// TIA Portal project "esteira_rejeito" (V16)
// primeiro projeto para o rejeito

(* hardware
DEVICE "S7-1200 station_1"  S7-1200 Station
   slot 0: "Rack_0"  S7-1200 Rack  Rack  V1.0
   slot 1: "PLC_1"  CPU 1212C DC/DC/DC  6ES7 212-1AE40-0XB0  V4.4
DEVICE "HMI_1"  KTP400 Basic PN
   slot 0: "HMI_1"  KTP400 Basic PN  6AV2 123-2DB03-0AX0  16.0.0.0
   slot 1: "HMI_RT_1"  KTP400 Basic PN  6AV2 123-2DB03-0AX0  16.0.0.0
   slot 5: "HMI_1.IE_CP_1"  PROFINET Interface  16.0.0.0
      slot 1: "PROFINET Interface_1"  PROFINET Interface
         slot 1: "Port_1"  Port
*)

// ===== PLC "PLC_1"  CPU 1212C DC/DC/DC =====

VAR_GLOBAL   // PLC tag table "Default tag table"
   "encoder_bk10_2101" AT %ID1000 : DInt;
   "ativa motor_bk10_2101" AT %M0.1 : Bool;
   "ativa motor_bk10_2101(1)" AT %Q0.0 : Bool;
   "sensor_01" AT %I0.1 : Bool;
   "sensor_02" AT %I0.2 : Bool;
   "set rest" AT %M0.2 : Bool;
   "b1 liga manual" AT %I0.3 : Bool;
   "rej_01" AT %M0.3 : Bool;
   "rej_01(1)" AT %M0.4 : Bool;
   "sensor_04" AT %I0.4 : Bool;
   "sensor_05" AT %I0.5 : Bool;
   "sensor_06" AT %I0.6 : Bool;
   "ativa motor_rej_01" AT %Q0.1 : Bool;
   "ativa motor_rej_02" AT %Q0.2 : Bool;
   "ativa motor_rej_03" AT %Q0.3 : Bool;
   "sinaleiro_L01" AT %Q0.4 : Bool;
   "rej_02" AT %M0.5 : Bool;
   "rej_02(2)" AT %M0.6 : Bool;
   "rej_03" AT %M0.7 : Bool;
   "rej_03(1)" AT %M1.0 : Bool;
END_VAR

// folder: System blocks/Program resources

DATA_BLOCK "db_rej_01"   // DB3
{ S7_Optimized_Access := 'TRUE' }
AUTHOR : Simatic
FAMILY : IEC
NAME : IEC_TMR
VERSION : 1.0
// stored: InstanceOfName IEC_TIMER
"IEC_TIMER"
BEGIN
END_DATA_BLOCK

DATA_BLOCK "db_rej_02"   // DB4
{ S7_Optimized_Access := 'TRUE' }
AUTHOR : Simatic
FAMILY : IEC
NAME : IEC_TMR
VERSION : 1.0
// stored: InstanceOfName IEC_TIMER
"IEC_TIMER"
BEGIN
END_DATA_BLOCK

// folder: (top level)

FUNCTION "fc_bk10_2101" : Void   // FC2, LAD
{ S7_Optimized_Access := 'TRUE' }
VERSION : 0.1
   VAR_INPUT
      Input_1 : DInt;
   END_VAR
BEGIN

REGION Network 1
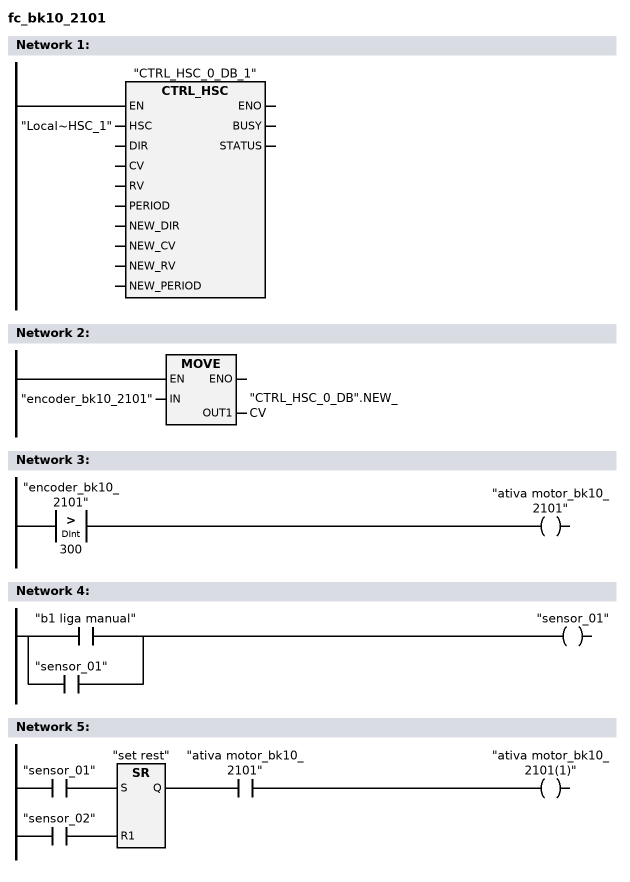
   "CTRL_HSC_0_DB_1"(HSC := "Local~HSC_1");   // CTRL_HSC
END_REGION

REGION Network 2
   RUNG wire#powerrail
      Move(in := "encoder_bk10_2101", out1 => "CTRL_HSC_0_DB".NEW_CV)
   END_RUNG
   // the same network as SCL:
   "CTRL_HSC_0_DB".NEW_CV := "encoder_bk10_2101";
END_REGION

REGION Network 3
   RUNG wire#powerrail
      { S7_Templates := "SrcType := DInt" } GT_Contact(in1 := "encoder_bk10_2101", in2 := 300)
      Coil( "ativa motor_bk10_2101" )
   END_RUNG
   // the same network as SCL:
   "ativa motor_bk10_2101" := "encoder_bk10_2101" > 300;
END_REGION

REGION Network 4
   RUNG wire#powerrail
      Contact( "b1 liga manual" )
      wire#w1
      Coil( "sensor_01" )
   END_RUNG
   RUNG wire#powerrail
      Contact( "sensor_01" )
   END_RUNG wire#w1
   // the same network as SCL:
   "sensor_01" := "b1 liga manual" OR "sensor_01";
END_REGION

REGION Network 5
   RUNG wire#powerrail
      Contact( "sensor_01" )
      S_SR(operand := "set rest", r1 := wire#w1)
      Contact( "ativa motor_bk10_2101" )
      Coil( "ativa motor_bk10_2101(1)" )
   END_RUNG
   RUNG wire#powerrail
      Contact( "sensor_02" )
   END_RUNG wire#w1
   // the same network as SCL:
   IF "sensor_01" THEN
       "set rest" := TRUE;   // SR flip-flop
   END_IF;
   IF "sensor_02" THEN "set rest" := FALSE; END_IF;
   "ativa motor_bk10_2101(1)" := "set rest" AND "ativa motor_bk10_2101";
END_REGION
END_FUNCTION

FUNCTION "fc_rej_01" : Void   // FC3, LAD
{ S7_Optimized_Access := 'TRUE' }
VERSION : 0.1
   VAR_TEMP   // added for the SCL form of the ladder/FBD networks
      _w1 : Bool;
   END_VAR
BEGIN

REGION Network 1
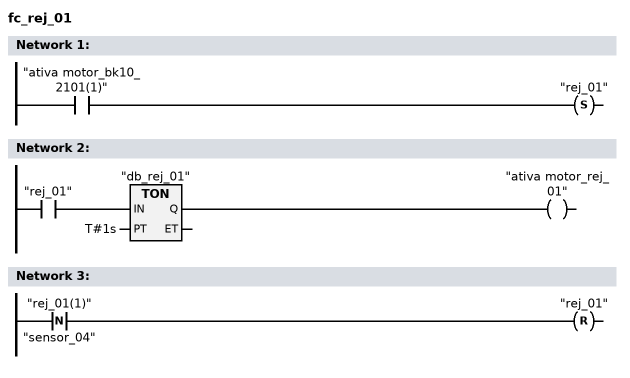
   RUNG wire#powerrail
      Contact( "ativa motor_bk10_2101(1)" )
      S_Coil( "rej_01" )
   END_RUNG
   // the same network as SCL:
   IF "ativa motor_bk10_2101(1)" THEN "rej_01" := TRUE; END_IF;
END_REGION

REGION Network 2
   "db_rej_01".TON(IN := "rej_01", PT := T#1s);
   "ativa motor_rej_01" := "db_rej_01".Q;
END_REGION

REGION Network 3
   RUNG wire#powerrail
      N_Contact(operand := "rej_01(1)", bit := "sensor_04")
      R_Coil( "rej_01" )
   END_RUNG
   // the same network as SCL:
   #_w1 := NOT "rej_01(1)" AND "sensor_04";   // falling edge of "rej_01(1)"
   "sensor_04" := "rej_01(1)";
   IF #_w1 THEN "rej_01" := FALSE; END_IF;
END_REGION
END_FUNCTION

FUNCTION "fc_rej_04" : Void   // FC4, LAD
{ S7_Optimized_Access := 'TRUE' }
VERSION : 0.1
   VAR_TEMP   // added for the SCL form of the ladder/FBD networks
      _w1 : Bool;
   END_VAR
BEGIN

REGION Network 1
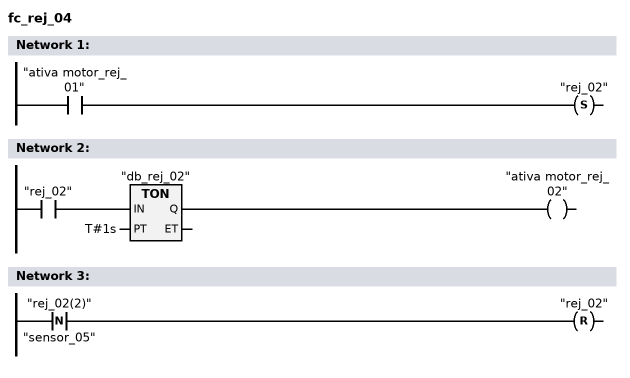
   RUNG wire#powerrail
      Contact( "ativa motor_rej_01" )
      S_Coil( "rej_02" )
   END_RUNG
   // the same network as SCL:
   IF "ativa motor_rej_01" THEN "rej_02" := TRUE; END_IF;
END_REGION

REGION Network 2
   "db_rej_02".TON(IN := "rej_02", PT := T#1s);
   "ativa motor_rej_02" := "db_rej_02".Q;
END_REGION

REGION Network 3
   RUNG wire#powerrail
      N_Contact(operand := "rej_02(2)", bit := "sensor_05")
      R_Coil( "rej_02" )
   END_RUNG
   // the same network as SCL:
   #_w1 := NOT "rej_02(2)" AND "sensor_05";   // falling edge of "rej_02(2)"
   "sensor_05" := "rej_02(2)";
   IF #_w1 THEN "rej_02" := FALSE; END_IF;
END_REGION
END_FUNCTION

ORGANIZATION_BLOCK "Main"   // OB1, LAD, ProgramCycle
TITLE = "Main Program Sweep (Cycle)"
{ S7_Optimized_Access := 'TRUE' }
VERSION : 0.1
   VAR_INPUT
      Initial_Call : Bool;   // Initial call of this OB
      Remanence : Bool;   // =True, if remanent data are available
   END_VAR
BEGIN
END_ORGANIZATION_BLOCK

ORGANIZATION_BLOCK "ob_bk10_2101"   // OB123, LAD, ProgramCycle
TITLE = "Main Program Sweep (Cycle)"
{ S7_Optimized_Access := 'TRUE' }
VERSION : 0.1
   VAR_INPUT
      Initial_Call : Bool;   // Initial call of this OB
      Remanence : Bool;   // =True, if remanent data are available
   END_VAR
BEGIN

REGION Network 1
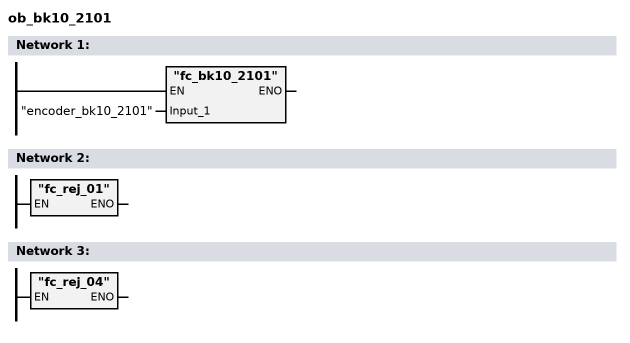
   RUNG wire#powerrail
      "fc_bk10_2101"(Input_1 := "encoder_bk10_2101")
   END_RUNG
   // the same network as SCL:
   "fc_bk10_2101"(Input_1 := "encoder_bk10_2101");
END_REGION

REGION Network 2
   RUNG wire#powerrail
      "fc_rej_01"()
   END_RUNG
   // the same network as SCL:
   "fc_rej_01"();
END_REGION

REGION Network 3
   RUNG wire#powerrail
      "fc_rej_04"()
   END_RUNG
   // the same network as SCL:
   "fc_rej_04"();
END_REGION
END_ORGANIZATION_BLOCK

(* ===== HMI "HMI_RT_1" =====
system functions are stored by id; their names below are inferred from use

HMI tags "Default tag table"
   "Tag_ScreenNumber" : UInt, internal

Template "Template_1" 480x272
   Button "Exit" at 388,227 size 63x44; TextOff 'Exit'; PictureOff "ExitRuntime_KTP400_Basic_PN_TR"; PictureOn "ExitRuntime_KTP400_Basic_PN_TR"
      on Release: StopRuntime(0)
   Button "Template_Button" at 268,227 size 63x44; TextOff 'Text'
   Button "Alarms" at 148,227 size 63x44; TextOff 'Alarms'; PictureOff "AlarmDisplay_KTP400_Basic_PN_TR"; PictureOn "AlarmDisplay_KTP400_Basic_PN_TR"
      on Release: function_ef3f5d25("Alarm window_Unacknowledged", -1)
   Button "Start screen" at 28,227 size 63x44; TextOff 'Start screen'; PictureOff "NavigateHome_KTP400_Basic_PN_TR"; PictureOn "NavigateHome_KTP400_Basic_PN_TR"
      on Release: ActivateScreen("Root screen", 0)
   SymbolicIOField "Symbolic_IO_Field_Screen" at 82,8 size 311x29; TextOff '0'; TextOn '1'; TextList "TextList_ScreenNames"
      ProcessValue <- "Tag_ScreenNumber"
      on Change: ActivateScreenByNumber("Tag_ScreenNumber", 0)
   DateTimeField "HmiScreenItemData" at 395,22 size 85x22
   DateTimeField "HmiScreenItemData_1" at 395,0 size 85x22
   GraphicView "Logo" at 0,0 size 80x45; Picture "Logo of HMI_1"

screen "Root screen" 480x272, template "Template_1"
   on GenerateScreen: SetTag("Tag_ScreenNumber", 1)
   TextField "HmiScreenItemData" at 48,122 size 384x22; Text 'Welcome to HMI_1 (KTP400 Basic+ PN)!'
*)